{attribute 'GeneratedUsingTerminal: EL1262-0000-0002'}
{attribute addProperty BoxType "EL1262-0000-0002"}
{attribute addProperty Id "Ch1_InputAT %I*BOOL1"}
{attribute addProperty CRC "4291087908"}
{attribute addProperty Size "1"}
TYPE Ch1_Input_FFC4CE24 EXTENDS InputBase_8311D824 :
STRUCT
	{attribute addProperty Name "Ch1_Input"}
	Ch1_Input AT %I* : BOOL;
END_STRUCT
END_TYPE

(* stored: Version 1.2.0.0, ProductVersion 3.1.4024.9
   DUT Ch1_Input_FFC4CE24: Id {b7d0ded0-a51c-43f2-b4c4-80487d99d4dc} *)
